(* PLC project Unnamed, Unknown Unnamed 1 *)
(* stored: creationDateTime 2023-04-09T20:23:42, modificationDateTime 2023-05-16T14:21:49 *)

PROGRAM Part1
  VAR_EXTERNAL
    START : BOOL;
    STOP : BOOL;
    CONR4_1 : BOOL;
    CONR4_2 : BOOL;
    SENDIF13 : BOOL;
  END_VAR
  VAR
    SENVIS1 AT %IX100.2 : BOOL;
    SENVIS2 AT %IX100.3 : BOOL;
    SENVIS3 AT %IX100.4 : BOOL;
    SENCAP2 AT %IX102.2 : BOOL;
    SENCAP3 AT %IX102.3 : BOOL;
    SENCAP5 AT %IX102.5 : BOOL;
    SENCAP6 AT %IX102.6 : BOOL;
    TTFrontLimit1 AT %IX103.0 : BOOL;
    TTFrontLimit2 AT %IX103.1 : BOOL;
    TTLimit90_1 AT %IX103.2 : BOOL;
    TTLimit90_2 AT %IX103.3 : BOOL;
    SENCAP8 AT %IX103.4 : BOOL;
    SENCAP9 AT %IX103.5 : BOOL;
    SENCAP10 AT %IX105.1 : BOOL;
    SENCAP11 AT %IX105.2 : BOOL;
    SENCAP12 AT %IX105.3 : BOOL;
    SENCAP13 AT %IX105.4 : BOOL;
    CON2_1 AT %QX100.0 : BOOL;
    CON2_2 AT %QX100.1 : BOOL;
    CON4_1 AT %QX100.2 : BOOL;
    CON4_2 AT %QX100.3 : BOOL;
    CON4_3 AT %QX100.4 : BOOL;
    CON6_1 AT %QX101.0 : BOOL;
    CON6_2 AT %QX101.1 : BOOL;
  END_VAR
  VAR_OUTPUT
    CON6_3 : BOOL;
    CON6_5 : BOOL;
    CON6_7 : BOOL;
  END_VAR
  VAR
    CONSCALE1 AT %QX102.0 : BOOL;
    CONSCALE2 AT %QX102.1 : BOOL;
    CONCURV1 AT %QX102.2 : BOOL;
    CONCURV2 AT %QX102.3 : BOOL;
    PIVOTARM1 AT %QX102.4 : BOOL;
    PIVOTARM2 AT %QX102.5 : BOOL;
    PIVOTARM3 AT %QX102.6 : BOOL;
    PIVOTURN1 AT %QX102.7 : BOOL;
    PIVOTURN2 AT %QX103.0 : BOOL;
    PIVOTURN3 AT %QX103.1 : BOOL;
    MCStart1 AT %QX103.2 : BOOL;
    MCStart2 AT %QX103.3 : BOOL;
    MCStart3 AT %QX103.4 : BOOL;
    MCStop1 AT %QX103.5 : BOOL;
    MCStop2 AT %QX103.6 : BOOL;
    MCStop3 AT %QX103.7 : BOOL;
    TurnTable1 AT %QX109.1 : BOOL;
    TurnTable2 AT %QX109.2 : BOOL;
    TTPles1 AT %QX109.3 : BOOL;
    TTPles2 AT %QX109.4 : BOOL;
    RollStop1 AT %QX109.5 : BOOL;
    RollStop2 AT %QX109.6 : BOOL;
    RollStop3 AT %QX109.7 : BOOL;
    RollStop4 AT %QX110.0 : BOOL;
    RollStop5 AT %QX110.1 : BOOL;
    RollStop6 AT %QX110.2 : BOOL;
  END_VAR
  VAR_EXTERNAL
    RollStop7 : BOOL;
  END_VAR
  VAR
    VIR1 AT %QX4.1 : BOOL;
    VIR2 AT %QX4.2 : BOOL;
    VIR10 AT %QX8.4 : BOOL;
    VIR11 AT %QX8.5 : BOOL;
  END_VAR
  VAR
    TOF1 : TOF;
    TOF2 : TOF;
    CTU0 : CTU;
  END_VAR
  VAR  (* added by the conversion: wires and edge detectors of the diagram *)
    R_TRIG1 : R_TRIG;
    R_TRIG2 : R_TRIG;
    R_TRIG3 : R_TRIG;
    R_TRIG4 : R_TRIG;
  END_VAR

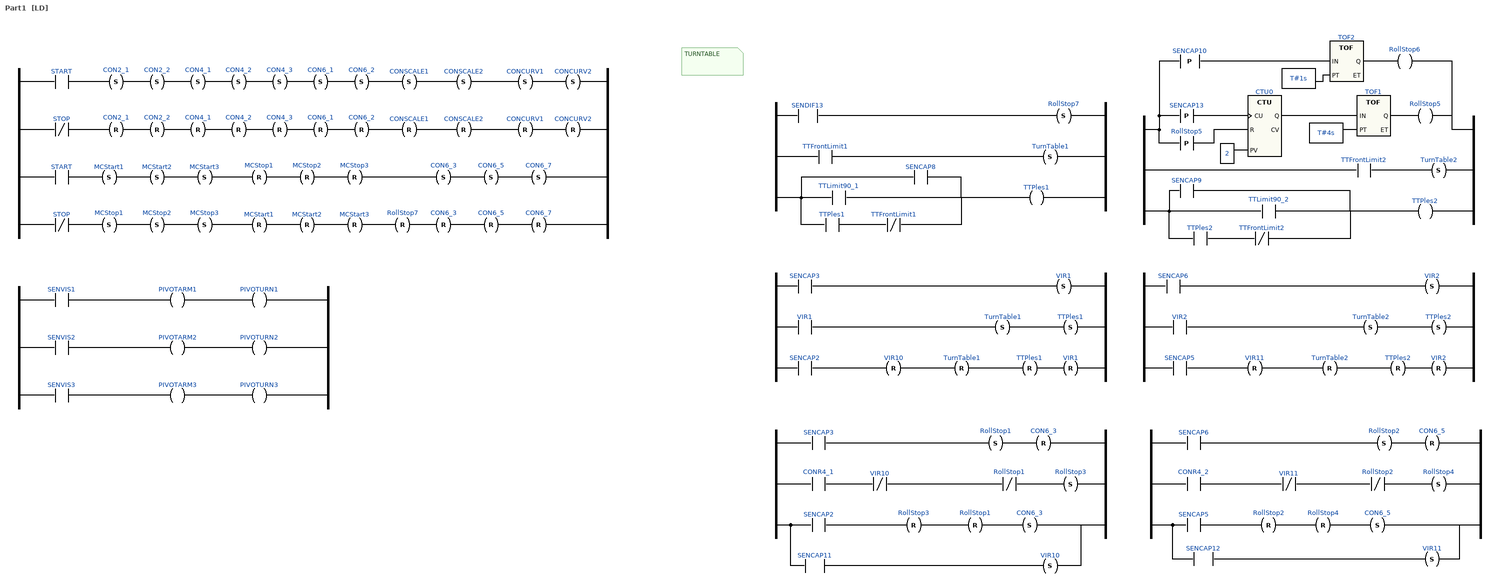
(* LD diagram, written out as Structured Text *)
(* TURNTABLE *)
R_TRIG1(CLK := SENCAP10);
TOF2(IN := R_TRIG1.Q, PT := T#1s);
RollStop6 := TOF2.Q;
IF START THEN CON2_1 := TRUE; END_IF;
IF START THEN CON2_2 := TRUE; END_IF;
IF START THEN CON4_1 := TRUE; END_IF;
IF START THEN CON4_2 := TRUE; END_IF;
IF START THEN CON4_3 := TRUE; END_IF;
IF START THEN CON6_1 := TRUE; END_IF;
IF START THEN CON6_2 := TRUE; END_IF;
IF START THEN CONSCALE1 := TRUE; END_IF;
IF START THEN CONSCALE2 := TRUE; END_IF;
IF START THEN CONCURV1 := TRUE; END_IF;
IF START THEN CONCURV2 := TRUE; END_IF;
IF SENDIF13 THEN RollStop7 := TRUE; END_IF;
R_TRIG2(CLK := SENCAP13);
R_TRIG3(CLK := R_TRIG2.Q);
R_TRIG4(CLK := RollStop5);
CTU0(CU := R_TRIG3.Q, R := R_TRIG4.Q, PV := 2);
TOF1(IN := CTU0.Q, PT := T#4s);
RollStop5 := TOF1.Q;
IF NOT STOP THEN CON2_1 := FALSE; END_IF;
IF NOT STOP THEN CON2_2 := FALSE; END_IF;
IF NOT STOP THEN CON4_1 := FALSE; END_IF;
IF NOT STOP THEN CON4_2 := FALSE; END_IF;
IF NOT STOP THEN CON4_3 := FALSE; END_IF;
IF NOT STOP THEN CON6_1 := FALSE; END_IF;
IF NOT STOP THEN CON6_2 := FALSE; END_IF;
IF NOT STOP THEN CONSCALE1 := FALSE; END_IF;
IF NOT STOP THEN CONSCALE2 := FALSE; END_IF;
IF NOT STOP THEN CONCURV1 := FALSE; END_IF;
IF NOT STOP THEN CONCURV2 := FALSE; END_IF;
IF TTFrontLimit1 THEN TurnTable1 := TRUE; END_IF;
IF TTFrontLimit2 THEN TurnTable2 := TRUE; END_IF;
IF START THEN MCStart1 := TRUE; END_IF;
IF START THEN MCStart2 := TRUE; END_IF;
IF START THEN MCStart3 := TRUE; END_IF;
IF START THEN MCStop1 := FALSE; END_IF;
IF START THEN MCStop2 := FALSE; END_IF;
IF START THEN MCStop3 := FALSE; END_IF;
IF START THEN CON6_3 := TRUE; END_IF;
IF START THEN CON6_5 := TRUE; END_IF;
IF START THEN CON6_7 := TRUE; END_IF;
TTPles1 := TTLimit90_1 OR SENCAP8 OR TTPles1 AND NOT TTFrontLimit1;
TTPles2 := TTLimit90_2 OR SENCAP9 OR TTPles2 AND NOT TTFrontLimit2;
IF NOT STOP THEN MCStop1 := TRUE; END_IF;
IF NOT STOP THEN MCStop2 := TRUE; END_IF;
IF NOT STOP THEN MCStop3 := TRUE; END_IF;
IF NOT STOP THEN MCStart1 := FALSE; END_IF;
IF NOT STOP THEN MCStart2 := FALSE; END_IF;
IF NOT STOP THEN MCStart3 := FALSE; END_IF;
IF NOT STOP THEN RollStop7 := FALSE; END_IF;
IF NOT STOP THEN CON6_3 := FALSE; END_IF;
IF NOT STOP THEN CON6_5 := FALSE; END_IF;
IF NOT STOP THEN CON6_7 := FALSE; END_IF;
IF SENCAP3 THEN VIR1 := TRUE; END_IF;
IF SENCAP6 THEN VIR2 := TRUE; END_IF;
PIVOTARM1 := SENVIS1;
PIVOTURN1 := SENVIS1;
IF VIR1 THEN TurnTable1 := TRUE; END_IF;
IF VIR1 THEN TTPles1 := TRUE; END_IF;
IF VIR2 THEN TurnTable2 := TRUE; END_IF;
IF VIR2 THEN TTPles2 := TRUE; END_IF;
PIVOTARM2 := SENVIS2;
PIVOTURN2 := SENVIS2;
IF SENCAP2 THEN VIR10 := FALSE; END_IF;
IF SENCAP2 THEN TurnTable1 := FALSE; END_IF;
IF SENCAP2 THEN TTPles1 := FALSE; END_IF;
IF SENCAP2 THEN VIR1 := FALSE; END_IF;
IF SENCAP5 THEN VIR11 := FALSE; END_IF;
IF SENCAP5 THEN TurnTable2 := FALSE; END_IF;
IF SENCAP5 THEN TTPles2 := FALSE; END_IF;
IF SENCAP5 THEN VIR2 := FALSE; END_IF;
PIVOTARM3 := SENVIS3;
PIVOTURN3 := SENVIS3;
IF SENCAP3 THEN RollStop1 := TRUE; END_IF;
IF SENCAP3 THEN CON6_3 := FALSE; END_IF;
IF SENCAP6 THEN RollStop2 := TRUE; END_IF;
IF SENCAP6 THEN CON6_5 := FALSE; END_IF;
IF CONR4_1 AND NOT VIR10 AND NOT RollStop1 THEN RollStop3 := TRUE; END_IF;
IF CONR4_2 AND NOT VIR11 AND NOT RollStop2 THEN RollStop4 := TRUE; END_IF;
IF SENCAP2 THEN RollStop3 := FALSE; END_IF;
IF SENCAP2 THEN RollStop1 := FALSE; END_IF;
IF SENCAP2 THEN CON6_3 := TRUE; END_IF;
IF SENCAP5 THEN RollStop2 := FALSE; END_IF;
IF SENCAP5 THEN RollStop4 := FALSE; END_IF;
IF SENCAP5 THEN CON6_5 := TRUE; END_IF;
IF SENCAP12 THEN VIR11 := TRUE; END_IF;
IF SENCAP11 THEN VIR10 := TRUE; END_IF;
END_PROGRAM

PROGRAM Part2
  VAR_EXTERNAL
    START : BOOL;
    STOP : BOOL;
  END_VAR
  VAR
    SENDIF1 AT %IX100.5 : BOOL;
    SENDIF2 AT %IX100.6 : BOOL;
    SENDIF5 AT %IX101.1 : BOOL;
    SENDIF6 AT %IX101.2 : BOOL;
    SENDIF9 AT %IX101.5 : BOOL;
    SENDIF10 AT %IX101.6 : BOOL;
    CON4_4 AT %QX100.5 : BOOL;
    CON4_5 AT %QX100.6 : BOOL;
    CON4_6 AT %QX100.7 : BOOL;
    CLAMP1 AT %QX104.0 : BOOL;
    CLAMP2 AT %QX104.1 : BOOL;
    CLAMP4 AT %QX104.3 : BOOL;
    CLAMP5 AT %QX104.4 : BOOL;
    CLAMP7 AT %QX104.6 : BOOL;
    CLAMP8 AT %QX104.7 : BOOL;
    RiseCLP1 AT %QX105.1 : BOOL;
    RiseCLP4 AT %QX105.2 : BOOL;
    RiseCLP7 AT %QX105.3 : BOOL;
    X1 AT %QX105.4 : BOOL;
    Z1 AT %QX105.5 : BOOL;
    GRAB1 AT %QX105.6 : BOOL;
    X2 AT %QX105.7 : BOOL;
    Z2 AT %QX106.0 : BOOL;
    GRAB2 AT %QX106.1 : BOOL;
    X3 AT %QX106.2 : BOOL;
    Z3 AT %QX106.3 : BOOL;
    GRAB3 AT %QX106.4 : BOOL;
    VIR1 AT %QX0.0 : BOOL;
    VIR2 AT %QX0.1 : BOOL;
    VIR3 AT %QX0.2 : BOOL;
    VIR4 AT %QX0.3 : BOOL;
    VIR5 AT %QX0.4 : BOOL;
    VIR6 AT %QX0.5 : BOOL;
    VIR7 AT %QX0.6 : BOOL;
    VIR8 AT %QX0.7 : BOOL;
    VIR9 AT %QX1.0 : BOOL;
    VIR10 AT %QX1.1 : BOOL;
    VIR11 AT %QX1.2 : BOOL;
    VIR12 AT %QX1.3 : BOOL;
  END_VAR
  VAR
    TON1 : TON;
    TON2 : TON;
    TON3 : TON;
    TON4 : TON;
    TON5 : TON;
    TON0 : TON;
    TON6 : TON;
    TON7 : TON;
    TON8 : TON;
    TON9 : TON;
    TON10 : TON;
    TON11 : TON;
    TON12 : TON;
    TON13 : TON;
    TON14 : TON;
    TON15 : TON;
    TON16 : TON;
    TON17 : TON;
    TON18 : TON;
    TON19 : TON;
    TON20 : TON;
  END_VAR

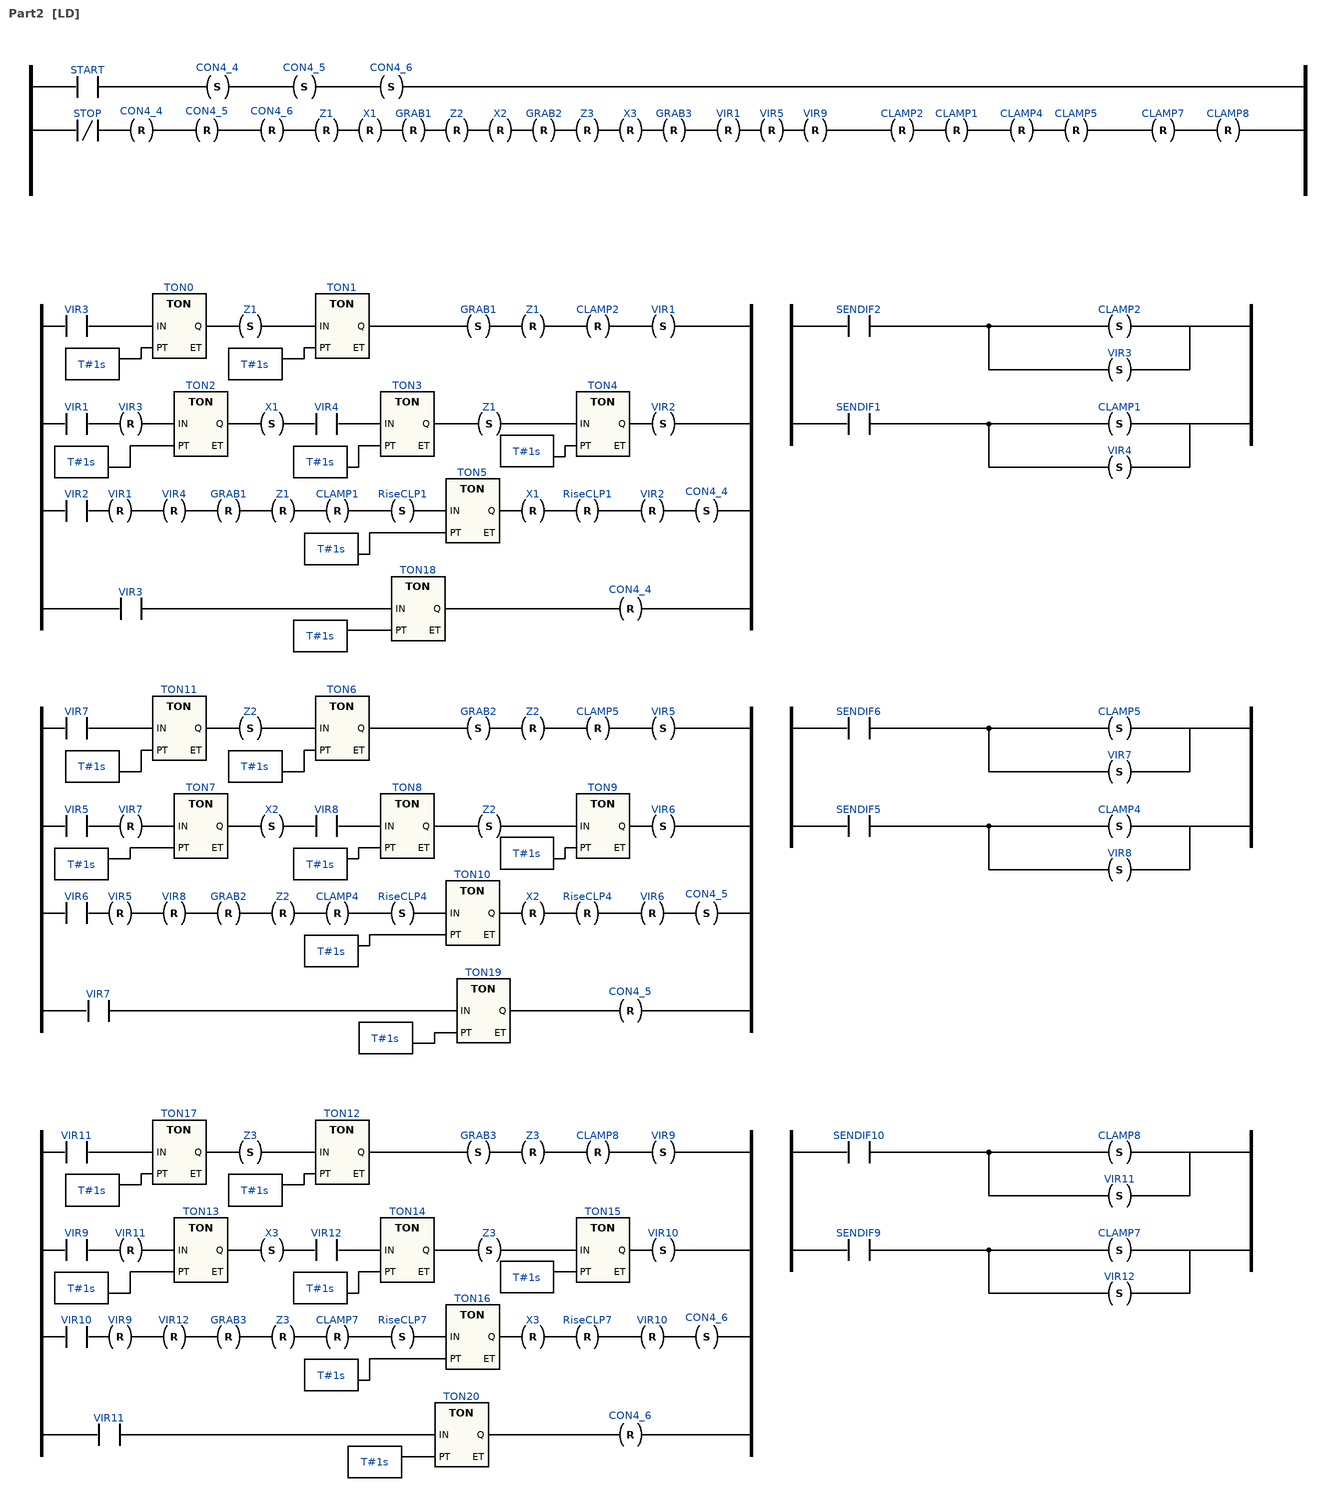
(* LD diagram, written out as Structured Text *)
IF START THEN CON4_4 := TRUE; END_IF;
IF START THEN CON4_5 := TRUE; END_IF;
IF START THEN CON4_6 := TRUE; END_IF;
IF NOT STOP THEN CON4_4 := FALSE; END_IF;
IF NOT STOP THEN CON4_5 := FALSE; END_IF;
IF NOT STOP THEN CON4_6 := FALSE; END_IF;
IF NOT STOP THEN Z1 := FALSE; END_IF;
IF NOT STOP THEN X1 := FALSE; END_IF;
IF NOT STOP THEN GRAB1 := FALSE; END_IF;
IF NOT STOP THEN Z2 := FALSE; END_IF;
IF NOT STOP THEN X2 := FALSE; END_IF;
IF NOT STOP THEN GRAB2 := FALSE; END_IF;
IF NOT STOP THEN Z3 := FALSE; END_IF;
IF NOT STOP THEN X3 := FALSE; END_IF;
IF NOT STOP THEN GRAB3 := FALSE; END_IF;
IF NOT STOP THEN VIR1 := FALSE; END_IF;
IF NOT STOP THEN VIR5 := FALSE; END_IF;
IF NOT STOP THEN VIR9 := FALSE; END_IF;
IF NOT STOP THEN CLAMP2 := FALSE; END_IF;
IF NOT STOP THEN CLAMP1 := FALSE; END_IF;
IF NOT STOP THEN CLAMP4 := FALSE; END_IF;
IF NOT STOP THEN CLAMP5 := FALSE; END_IF;
IF NOT STOP THEN CLAMP7 := FALSE; END_IF;
IF NOT STOP THEN CLAMP8 := FALSE; END_IF;
TON0(IN := VIR3, PT := T#1s);
IF TON0.Q THEN Z1 := TRUE; END_IF;
TON1(IN := TON0.Q, PT := T#1s);
IF TON1.Q THEN GRAB1 := TRUE; END_IF;
IF TON1.Q THEN Z1 := FALSE; END_IF;
IF TON1.Q THEN CLAMP2 := FALSE; END_IF;
IF TON1.Q THEN VIR1 := TRUE; END_IF;
IF SENDIF2 THEN CLAMP2 := TRUE; END_IF;
IF SENDIF2 THEN VIR3 := TRUE; END_IF;
IF VIR1 THEN VIR3 := FALSE; END_IF;
TON2(IN := VIR1, PT := T#1s);
IF TON2.Q THEN X1 := TRUE; END_IF;
TON3(IN := TON2.Q AND VIR4, PT := T#1s);
IF TON3.Q THEN Z1 := TRUE; END_IF;
TON4(IN := TON3.Q, PT := T#1s);
IF TON4.Q THEN VIR2 := TRUE; END_IF;
IF SENDIF1 THEN CLAMP1 := TRUE; END_IF;
IF SENDIF1 THEN VIR4 := TRUE; END_IF;
IF VIR2 THEN VIR1 := FALSE; END_IF;
IF VIR2 THEN VIR4 := FALSE; END_IF;
IF VIR2 THEN GRAB1 := FALSE; END_IF;
IF VIR2 THEN Z1 := FALSE; END_IF;
IF VIR2 THEN CLAMP1 := FALSE; END_IF;
IF VIR2 THEN RiseCLP1 := TRUE; END_IF;
TON5(IN := VIR2, PT := T#1s);
IF TON5.Q THEN X1 := FALSE; END_IF;
IF TON5.Q THEN RiseCLP1 := FALSE; END_IF;
IF TON5.Q THEN VIR2 := FALSE; END_IF;
IF TON5.Q THEN CON4_4 := TRUE; END_IF;
TON18(IN := VIR3, PT := T#1s);
IF TON18.Q THEN CON4_4 := FALSE; END_IF;
TON11(IN := VIR7, PT := T#1s);
IF TON11.Q THEN Z2 := TRUE; END_IF;
TON6(IN := TON11.Q, PT := T#1s);
IF TON6.Q THEN GRAB2 := TRUE; END_IF;
IF TON6.Q THEN Z2 := FALSE; END_IF;
IF TON6.Q THEN CLAMP5 := FALSE; END_IF;
IF TON6.Q THEN VIR5 := TRUE; END_IF;
IF SENDIF6 THEN CLAMP5 := TRUE; END_IF;
IF SENDIF6 THEN VIR7 := TRUE; END_IF;
IF VIR5 THEN VIR7 := FALSE; END_IF;
TON7(IN := VIR5, PT := T#1s);
IF TON7.Q THEN X2 := TRUE; END_IF;
TON8(IN := TON7.Q AND VIR8, PT := T#1s);
IF TON8.Q THEN Z2 := TRUE; END_IF;
TON9(IN := TON8.Q, PT := T#1s);
IF TON9.Q THEN VIR6 := TRUE; END_IF;
IF SENDIF5 THEN CLAMP4 := TRUE; END_IF;
IF SENDIF5 THEN VIR8 := TRUE; END_IF;
IF VIR6 THEN VIR5 := FALSE; END_IF;
IF VIR6 THEN VIR8 := FALSE; END_IF;
IF VIR6 THEN GRAB2 := FALSE; END_IF;
IF VIR6 THEN Z2 := FALSE; END_IF;
IF VIR6 THEN CLAMP4 := FALSE; END_IF;
IF VIR6 THEN RiseCLP4 := TRUE; END_IF;
TON10(IN := VIR6, PT := T#1s);
IF TON10.Q THEN X2 := FALSE; END_IF;
IF TON10.Q THEN RiseCLP4 := FALSE; END_IF;
IF TON10.Q THEN VIR6 := FALSE; END_IF;
IF TON10.Q THEN CON4_5 := TRUE; END_IF;
TON19(IN := VIR7, PT := T#1s);
IF TON19.Q THEN CON4_5 := FALSE; END_IF;
TON17(IN := VIR11, PT := T#1s);
IF TON17.Q THEN Z3 := TRUE; END_IF;
TON12(IN := TON17.Q, PT := T#1s);
IF TON12.Q THEN GRAB3 := TRUE; END_IF;
IF TON12.Q THEN Z3 := FALSE; END_IF;
IF TON12.Q THEN CLAMP8 := FALSE; END_IF;
IF TON12.Q THEN VIR9 := TRUE; END_IF;
IF SENDIF10 THEN CLAMP8 := TRUE; END_IF;
IF SENDIF10 THEN VIR11 := TRUE; END_IF;
IF VIR9 THEN VIR11 := FALSE; END_IF;
TON13(IN := VIR9, PT := T#1s);
IF TON13.Q THEN X3 := TRUE; END_IF;
TON14(IN := TON13.Q AND VIR12, PT := T#1s);
IF TON14.Q THEN Z3 := TRUE; END_IF;
TON15(IN := TON14.Q, PT := T#1s);
IF TON15.Q THEN VIR10 := TRUE; END_IF;
IF SENDIF9 THEN CLAMP7 := TRUE; END_IF;
IF SENDIF9 THEN VIR12 := TRUE; END_IF;
IF VIR10 THEN VIR9 := FALSE; END_IF;
IF VIR10 THEN VIR12 := FALSE; END_IF;
IF VIR10 THEN GRAB3 := FALSE; END_IF;
IF VIR10 THEN Z3 := FALSE; END_IF;
IF VIR10 THEN CLAMP7 := FALSE; END_IF;
IF VIR10 THEN RiseCLP7 := TRUE; END_IF;
TON16(IN := VIR10, PT := T#1s);
IF TON16.Q THEN X3 := FALSE; END_IF;
IF TON16.Q THEN RiseCLP7 := FALSE; END_IF;
IF TON16.Q THEN VIR10 := FALSE; END_IF;
IF TON16.Q THEN CON4_6 := TRUE; END_IF;
TON20(IN := VIR11, PT := T#1s);
IF TON20.Q THEN CON4_6 := FALSE; END_IF;
END_PROGRAM

PROGRAM Part3
  VAR_EXTERNAL
    START : BOOL;
    STOP : BOOL;
  END_VAR
  VAR
    SENDIF3 AT %IX100.7 : BOOL;
    SENDIF4 AT %IX101.0 : BOOL;
    SENDIF7 AT %IX101.3 : BOOL;
    SENDIF8 AT %IX101.4 : BOOL;
    SENDIF11 AT %IX101.7 : BOOL;
    SENDIF12 AT %IX102.0 : BOOL;
    SENCAP1 AT %IX102.1 : BOOL;
    SENCAP4 AT %IX102.4 : BOOL;
    SENCAP7 AT %IX102.7 : BOOL;
    CON6_4 AT %QX101.3 : BOOL;
    CON6_6 AT %QX101.5 : BOOL;
    CON6_8 AT %QX101.7 : BOOL;
    CLAMP3 AT %QX104.2 : BOOL;
    CLAMP6 AT %QX104.5 : BOOL;
    CLAMP9 AT %QX105.0 : BOOL;
    CW4 AT %QX106.5 : BOOL;
    CCW4 AT %QX106.6 : BOOL;
    CW5 AT %QX106.7 : BOOL;
    CCW5 AT %QX107.0 : BOOL;
    CW6 AT %QX107.1 : BOOL;
    CCW6 AT %QX107.2 : BOOL;
    GRAB4 AT %QX107.3 : BOOL;
    GRAB5 AT %QX107.4 : BOOL;
    GRAB6 AT %QX107.5 : BOOL;
    CONR2_1 AT %QX107.6 : BOOL;
    CONR2_2 AT %QX107.7 : BOOL;
    CONR2_3 AT %QX108.0 : BOOL;
  END_VAR
  VAR_EXTERNAL
    CONR4_1 : BOOL;
    CONR4_2 : BOOL;
  END_VAR
  VAR
    CONR4_3 AT %QX108.3 : BOOL;
    CONR4_4 AT %QX108.4 : BOOL;
    CONR6_1 AT %QX108.5 : BOOL;
    CONR6_2 AT %QX108.6 : BOOL;
    CONRLCCW1 AT %QX108.7 : BOOL;
    CONRLCCW2 AT %QX109.0 : BOOL;
    CLPRise3 AT %QX112.2 : BOOL;
    CLPRise6 AT %QX112.3 : BOOL;
    CLPRise9 AT %QX112.4 : BOOL;
    X4 AT %QW100 : INT;
    Z4 AT %QW101 : INT;
    X5 AT %QW102 : INT;
    Z5 AT %QW103 : INT;
    X6 AT %QW104 : INT;
    Z6 AT %QW105 : INT;
    VIR1 AT %QX1.4 : BOOL;
    VIR2 AT %QX1.5 : BOOL;
    VIR3 AT %QX1.6 : BOOL;
    VIR4 AT %QX1.7 : BOOL;
    VIR5 AT %QX2.0 : BOOL;
    VIR6 AT %QX2.1 : BOOL;
    VIR7 AT %QX2.2 : BOOL;
    VIR8 AT %QX2.3 : BOOL;
    VIR9 AT %QX2.4 : BOOL;
    VIR10 AT %QX2.5 : BOOL;
    VIR11 AT %QX2.6 : BOOL;
    VIR12 AT %QX2.7 : BOOL;
    VIR13 AT %QX3.0 : BOOL;
    VIR14 AT %QX3.1 : BOOL;
    VIR15 AT %QX3.2 : BOOL;
    VIR16 AT %QX3.3 : BOOL;
    VIR17 AT %QX3.4 : BOOL;
    VIR18 AT %QX3.5 : BOOL;
    VIR19 AT %QX3.6 : BOOL;
    VIR20 AT %QX3.7 : BOOL;
    VIR21 AT %QX4.0 : BOOL;
    VIR22 AT %QX5.6 : BOOL;
    VIR23 AT %QX5.7 : BOOL;
  END_VAR
  VAR_EXTERNAL
    CON6_3 : BOOL;
    CON6_5 : BOOL;
    CON6_7 : BOOL;
  END_VAR
  VAR
    TON0 : TON;
    TON1 : TON;
    TON2 : TON;
    TON3 : TON;
    TON4 : TON;
    TON5 : TON;
    TON6 : TON;
    TON7 : TON;
    TON8 : TON;
    TON9 : TON;
    TON10 : TON;
    TON11 : TON;
    TON12 : TON;
    TON13 : TON;
    TON14 : TON;
    TON15 : TON;
    TON16 : TON;
    CTU0 : CTU;
    TON17 : TON;
    TON18 : TON;
    TON19 : TON;
    TON20 : TON;
    TON21 : TON;
    TON22 : TON;
    TON23 : TON;
    TON24 : TON;
    TON25 : TON;
    TON26 : TON;
    TON27 : TON;
    TON28 : TON;
    TON29 : TON;
    TON30 : TON;
    TON31 : TON;
    TON32 : TON;
    TON33 : TON;
    CTU1 : CTU;
    TON34 : TON;
    TON35 : TON;
    TON36 : TON;
    TON37 : TON;
    TON38 : TON;
    TON39 : TON;
    TON40 : TON;
    TON41 : TON;
    TON42 : TON;
    TON43 : TON;
    TON44 : TON;
    TON45 : TON;
    TON46 : TON;
    TON47 : TON;
    TON48 : TON;
    TON49 : TON;
    TON50 : TON;
    CTU2 : CTU;
    TON51 : TON;
    TON52 : TON;
    TON53 : TON;
  END_VAR
  VAR  (* added by the conversion: wires and edge detectors of the diagram *)
    _MOVE66_ENO : BOOL;
    _MOVE66_OUT : INT;
    _MOVE25_ENO : BOOL;
    _MOVE25_OUT : INT;
    _MOVE288_ENO : BOOL;
    _MOVE288_OUT : INT;
    _MOVE249_ENO : BOOL;
    _MOVE249_OUT : INT;
    _MOVE44_ENO : BOOL;
    _MOVE44_OUT : INT;
    _MOVE51_ENO : BOOL;
    _MOVE51_OUT : INT;
    _MOVE268_ENO : BOOL;
    _MOVE268_OUT : INT;
    _MOVE275_ENO : BOOL;
    _MOVE275_OUT : INT;
    _MOVE73_ENO : BOOL;
    _MOVE73_OUT : INT;
    _MOVE76_ENO : BOOL;
    _MOVE76_OUT : INT;
    _MOVE83_ENO : BOOL;
    _MOVE83_OUT : INT;
    _MOVE295_ENO : BOOL;
    _MOVE295_OUT : INT;
    _MOVE298_ENO : BOOL;
    _MOVE298_OUT : INT;
    _MOVE305_ENO : BOOL;
    _MOVE305_OUT : INT;
    _MOVE89_ENO : BOOL;
    _MOVE89_OUT : INT;
    _MOVE94_ENO : BOOL;
    _MOVE94_OUT : INT;
    _MOVE311_ENO : BOOL;
    _MOVE311_OUT : INT;
    _MOVE316_ENO : BOOL;
    _MOVE316_OUT : INT;
    _MOVE100_ENO : BOOL;
    _MOVE100_OUT : INT;
    _MOVE322_ENO : BOOL;
    _MOVE322_OUT : INT;
    R_TRIG1 : R_TRIG;
    R_TRIG2 : R_TRIG;
    _MOVE177_ENO : BOOL;
    _MOVE177_OUT : INT;
    _MOVE138_ENO : BOOL;
    _MOVE138_OUT : INT;
    _MOVE157_ENO : BOOL;
    _MOVE157_OUT : INT;
    _MOVE164_ENO : BOOL;
    _MOVE164_OUT : INT;
    _MOVE184_ENO : BOOL;
    _MOVE184_OUT : INT;
    _MOVE187_ENO : BOOL;
    _MOVE187_OUT : INT;
    _MOVE194_ENO : BOOL;
    _MOVE194_OUT : INT;
    _MOVE200_ENO : BOOL;
    _MOVE200_OUT : INT;
    _MOVE205_ENO : BOOL;
    _MOVE205_OUT : INT;
    _MOVE211_ENO : BOOL;
    _MOVE211_OUT : INT;
    R_TRIG3 : R_TRIG;
  END_VAR

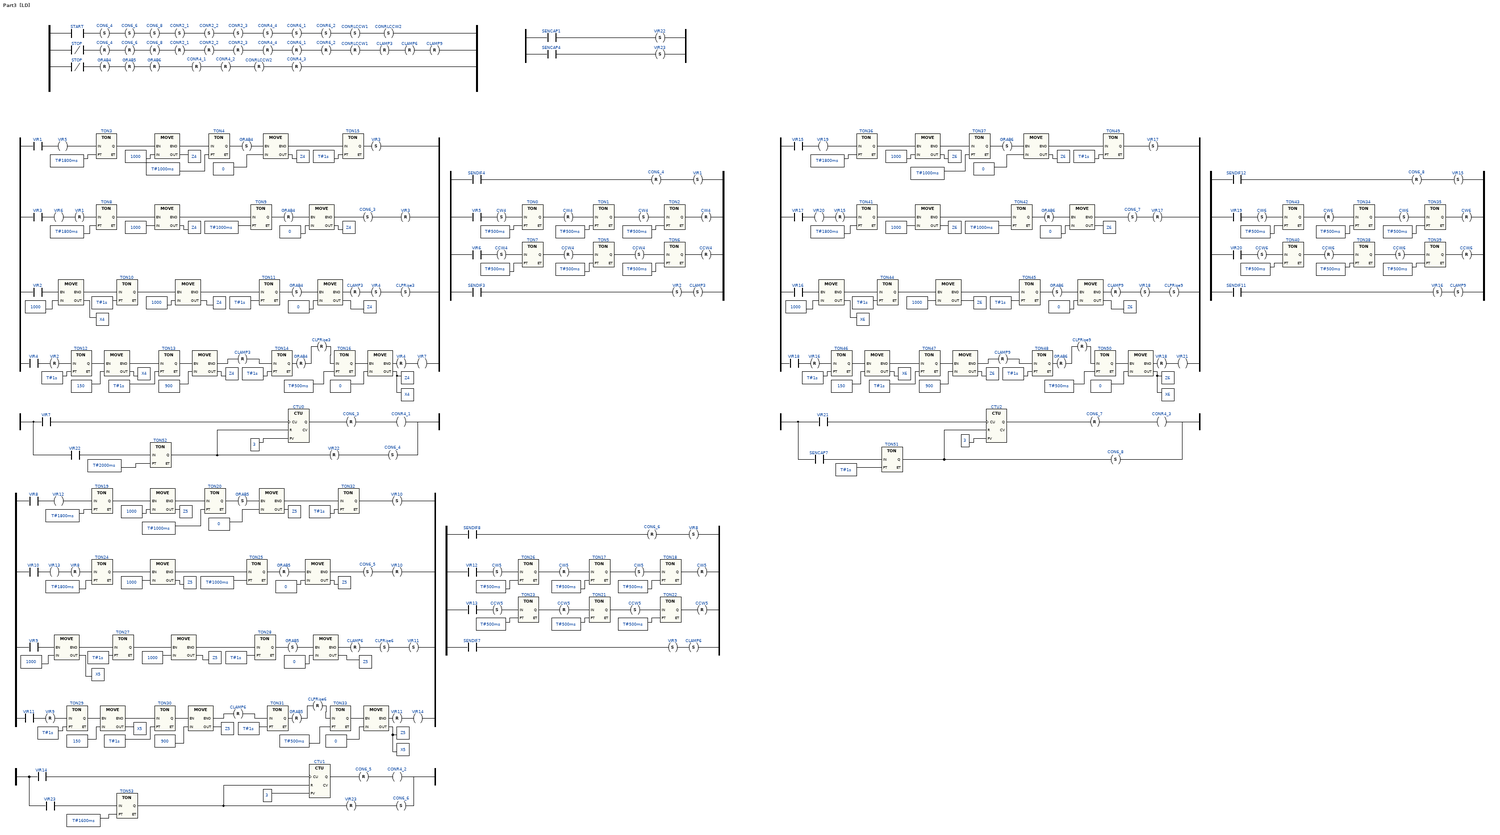
(* LD diagram, written out as Structured Text *)
IF START THEN CON6_4 := TRUE; END_IF;
IF START THEN CON6_6 := TRUE; END_IF;
IF START THEN CON6_8 := TRUE; END_IF;
IF START THEN CONR2_1 := TRUE; END_IF;
IF START THEN CONR2_2 := TRUE; END_IF;
IF START THEN CONR2_3 := TRUE; END_IF;
IF START THEN CONR4_4 := TRUE; END_IF;
IF START THEN CONR6_1 := TRUE; END_IF;
IF START THEN CONR6_2 := TRUE; END_IF;
IF START THEN CONRLCCW1 := TRUE; END_IF;
IF START THEN CONRLCCW2 := TRUE; END_IF;
IF SENCAP1 THEN VIR22 := TRUE; END_IF;
IF NOT STOP THEN CON6_4 := FALSE; END_IF;
IF NOT STOP THEN CON6_6 := FALSE; END_IF;
IF NOT STOP THEN CON6_8 := FALSE; END_IF;
IF NOT STOP THEN CONR2_1 := FALSE; END_IF;
IF NOT STOP THEN CONR2_2 := FALSE; END_IF;
IF NOT STOP THEN CONR2_3 := FALSE; END_IF;
IF NOT STOP THEN CONR4_4 := FALSE; END_IF;
IF NOT STOP THEN CONR6_1 := FALSE; END_IF;
IF NOT STOP THEN CONR6_2 := FALSE; END_IF;
IF NOT STOP THEN CONRLCCW1 := FALSE; END_IF;
IF NOT STOP THEN CLAMP3 := FALSE; END_IF;
IF NOT STOP THEN CLAMP6 := FALSE; END_IF;
IF NOT STOP THEN CLAMP9 := FALSE; END_IF;
IF SENCAP4 THEN VIR23 := TRUE; END_IF;
IF NOT STOP THEN GRAB4 := FALSE; END_IF;
IF NOT STOP THEN GRAB5 := FALSE; END_IF;
IF NOT STOP THEN GRAB6 := FALSE; END_IF;
IF NOT STOP THEN CONR4_1 := FALSE; END_IF;
IF NOT STOP THEN CONR4_2 := FALSE; END_IF;
IF NOT STOP THEN CONRLCCW2 := FALSE; END_IF;
IF NOT STOP THEN CONR4_3 := FALSE; END_IF;
VIR5 := VIR1;
TON3(IN := VIR1, PT := T#1800ms);
_MOVE66_OUT := MOVE(EN := TON3.Q, IN := 1000, ENO => _MOVE66_ENO);
TON4(IN := _MOVE66_ENO, PT := T#1000ms);
IF TON4.Q THEN GRAB4 := TRUE; END_IF;
_MOVE25_OUT := MOVE(EN := TON4.Q, IN := 0, ENO => _MOVE25_ENO);
TON15(IN := _MOVE25_ENO, PT := T#1s);
IF TON15.Q THEN VIR3 := TRUE; END_IF;
VIR19 := VIR15;
TON36(IN := VIR15, PT := T#1800ms);
_MOVE288_OUT := MOVE(EN := TON36.Q, IN := 1000, ENO => _MOVE288_ENO);
TON37(IN := _MOVE288_ENO, PT := T#1000ms);
IF TON37.Q THEN GRAB6 := TRUE; END_IF;
_MOVE249_OUT := MOVE(EN := TON37.Q, IN := 0, ENO => _MOVE249_ENO);
TON49(IN := _MOVE249_ENO, PT := T#1s);
IF TON49.Q THEN VIR17 := TRUE; END_IF;
IF _MOVE66_ENO THEN Z4 := _MOVE66_OUT; END_IF;
IF _MOVE25_ENO THEN Z4 := _MOVE25_OUT; END_IF;
IF _MOVE288_ENO THEN Z6 := _MOVE288_OUT; END_IF;
IF _MOVE249_ENO THEN Z6 := _MOVE249_OUT; END_IF;
IF SENDIF4 THEN CON6_4 := FALSE; END_IF;
IF SENDIF4 THEN VIR1 := TRUE; END_IF;
IF SENDIF12 THEN CON6_8 := FALSE; END_IF;
IF SENDIF12 THEN VIR15 := TRUE; END_IF;
VIR6 := VIR3;
IF VIR3 THEN VIR1 := FALSE; END_IF;
TON8(IN := VIR3, PT := T#1800ms);
_MOVE44_OUT := MOVE(EN := TON8.Q, IN := 1000, ENO => _MOVE44_ENO);
TON9(IN := _MOVE44_ENO, PT := T#1000ms);
IF TON9.Q THEN GRAB4 := FALSE; END_IF;
_MOVE51_OUT := MOVE(EN := TON9.Q, IN := 0, ENO => _MOVE51_ENO);
IF _MOVE51_ENO THEN CON6_3 := TRUE; END_IF;
IF _MOVE51_ENO THEN VIR3 := FALSE; END_IF;
IF VIR5 THEN CW4 := TRUE; END_IF;
TON0(IN := VIR5, PT := T#500ms);
IF TON0.Q THEN CW4 := FALSE; END_IF;
TON1(IN := TON0.Q, PT := T#500ms);
IF TON1.Q THEN CW4 := TRUE; END_IF;
TON2(IN := TON1.Q, PT := T#500ms);
IF TON2.Q THEN CW4 := FALSE; END_IF;
VIR20 := VIR17;
IF VIR17 THEN VIR15 := FALSE; END_IF;
TON41(IN := VIR17, PT := T#1800ms);
_MOVE268_OUT := MOVE(EN := TON41.Q, IN := 1000, ENO => _MOVE268_ENO);
TON42(IN := _MOVE268_ENO, PT := T#1000ms);
IF TON42.Q THEN GRAB6 := FALSE; END_IF;
_MOVE275_OUT := MOVE(EN := TON42.Q, IN := 0, ENO => _MOVE275_ENO);
IF _MOVE275_ENO THEN CON6_7 := TRUE; END_IF;
IF _MOVE275_ENO THEN VIR17 := FALSE; END_IF;
IF VIR19 THEN CW6 := TRUE; END_IF;
TON43(IN := VIR19, PT := T#500ms);
IF TON43.Q THEN CW6 := FALSE; END_IF;
TON34(IN := TON43.Q, PT := T#500ms);
IF TON34.Q THEN CW6 := TRUE; END_IF;
TON35(IN := TON34.Q, PT := T#500ms);
IF TON35.Q THEN CW6 := FALSE; END_IF;
IF _MOVE44_ENO THEN Z4 := _MOVE44_OUT; END_IF;
IF _MOVE51_ENO THEN Z4 := _MOVE51_OUT; END_IF;
IF _MOVE268_ENO THEN Z6 := _MOVE268_OUT; END_IF;
IF _MOVE275_ENO THEN Z6 := _MOVE275_OUT; END_IF;
IF VIR6 THEN CCW4 := TRUE; END_IF;
TON7(IN := VIR6, PT := T#500ms);
IF TON7.Q THEN CCW4 := FALSE; END_IF;
TON5(IN := TON7.Q, PT := T#500ms);
IF TON5.Q THEN CCW4 := TRUE; END_IF;
TON6(IN := TON5.Q, PT := T#500ms);
IF TON6.Q THEN CCW4 := FALSE; END_IF;
IF VIR20 THEN CCW6 := TRUE; END_IF;
TON40(IN := VIR20, PT := T#500ms);
IF TON40.Q THEN CCW6 := FALSE; END_IF;
TON38(IN := TON40.Q, PT := T#500ms);
IF TON38.Q THEN CCW6 := TRUE; END_IF;
TON39(IN := TON38.Q, PT := T#500ms);
IF TON39.Q THEN CCW6 := FALSE; END_IF;
_MOVE73_OUT := MOVE(EN := VIR2, IN := 1000, ENO => _MOVE73_ENO);
TON10(IN := _MOVE73_ENO, PT := T#1s);
_MOVE76_OUT := MOVE(EN := TON10.Q, IN := 1000, ENO => _MOVE76_ENO);
TON11(IN := _MOVE76_ENO, PT := T#1s);
IF TON11.Q THEN GRAB4 := TRUE; END_IF;
_MOVE83_OUT := MOVE(EN := TON11.Q, IN := 0, ENO => _MOVE83_ENO);
IF _MOVE83_ENO THEN CLAMP3 := FALSE; END_IF;
IF _MOVE83_ENO THEN VIR4 := TRUE; END_IF;
IF _MOVE83_ENO THEN CLPRise3 := TRUE; END_IF;
IF SENDIF3 THEN VIR2 := TRUE; END_IF;
IF SENDIF3 THEN CLAMP3 := TRUE; END_IF;
_MOVE295_OUT := MOVE(EN := VIR16, IN := 1000, ENO => _MOVE295_ENO);
TON44(IN := _MOVE295_ENO, PT := T#1s);
_MOVE298_OUT := MOVE(EN := TON44.Q, IN := 1000, ENO => _MOVE298_ENO);
TON45(IN := _MOVE298_ENO, PT := T#1s);
IF TON45.Q THEN GRAB6 := TRUE; END_IF;
_MOVE305_OUT := MOVE(EN := TON45.Q, IN := 0, ENO => _MOVE305_ENO);
IF _MOVE305_ENO THEN CLAMP9 := FALSE; END_IF;
IF _MOVE305_ENO THEN VIR18 := TRUE; END_IF;
IF _MOVE305_ENO THEN CLPRise9 := TRUE; END_IF;
IF SENDIF11 THEN VIR16 := TRUE; END_IF;
IF SENDIF11 THEN CLAMP9 := TRUE; END_IF;
IF _MOVE76_ENO THEN Z4 := _MOVE76_OUT; END_IF;
IF _MOVE298_ENO THEN Z6 := _MOVE298_OUT; END_IF;
IF _MOVE83_ENO THEN Z4 := _MOVE83_OUT; END_IF;
IF _MOVE305_ENO THEN Z6 := _MOVE305_OUT; END_IF;
IF _MOVE73_ENO THEN X4 := _MOVE73_OUT; END_IF;
IF _MOVE295_ENO THEN X6 := _MOVE295_OUT; END_IF;
TON12(IN := VIR4, PT := T#1s);
_MOVE89_OUT := MOVE(EN := TON12.Q, IN := 150, ENO => _MOVE89_ENO);
TON13(IN := _MOVE89_ENO, PT := T#1s);
_MOVE94_OUT := MOVE(EN := TON13.Q, IN := 900, ENO => _MOVE94_ENO);
TON14(IN := _MOVE94_ENO, PT := T#1s);
IF TON14.Q THEN CLPRise3 := FALSE; END_IF;
TON46(IN := VIR18, PT := T#1s);
_MOVE311_OUT := MOVE(EN := TON46.Q, IN := 150, ENO => _MOVE311_ENO);
TON47(IN := _MOVE311_ENO, PT := T#1s);
_MOVE316_OUT := MOVE(EN := TON47.Q, IN := 900, ENO => _MOVE316_ENO);
TON48(IN := _MOVE316_ENO, PT := T#1s);
IF TON48.Q THEN CLPRise9 := FALSE; END_IF;
IF _MOVE94_ENO THEN CLAMP3 := FALSE; END_IF;
IF _MOVE316_ENO THEN CLAMP9 := FALSE; END_IF;
IF VIR4 THEN VIR2 := FALSE; END_IF;
IF TON14.Q THEN GRAB4 := FALSE; END_IF;
TON16(IN := TON14.Q, PT := T#500ms);
_MOVE100_OUT := MOVE(EN := TON16.Q, IN := 0, ENO => _MOVE100_ENO);
IF _MOVE100_ENO THEN VIR4 := FALSE; END_IF;
VIR7 := _MOVE100_ENO;
IF VIR18 THEN VIR16 := FALSE; END_IF;
IF TON48.Q THEN GRAB6 := FALSE; END_IF;
TON50(IN := TON48.Q, PT := T#500ms);
_MOVE322_OUT := MOVE(EN := TON50.Q, IN := 0, ENO => _MOVE322_ENO);
IF _MOVE322_ENO THEN VIR18 := FALSE; END_IF;
VIR21 := _MOVE322_ENO;
IF _MOVE89_ENO THEN X4 := _MOVE89_OUT; END_IF;
IF _MOVE94_ENO THEN Z4 := _MOVE94_OUT; END_IF;
IF _MOVE311_ENO THEN X6 := _MOVE311_OUT; END_IF;
IF _MOVE316_ENO THEN Z6 := _MOVE316_OUT; END_IF;
IF _MOVE100_ENO THEN Z4 := _MOVE100_OUT; END_IF;
IF _MOVE322_ENO THEN Z6 := _MOVE322_OUT; END_IF;
IF _MOVE100_ENO THEN X4 := _MOVE100_OUT; END_IF;
IF _MOVE322_ENO THEN X6 := _MOVE322_OUT; END_IF;
R_TRIG1(CLK := VIR7);
TON52(IN := VIR22, PT := T#2000ms);
CTU0(CU := R_TRIG1.Q, R := TON52.Q, PV := 3);
IF CTU0.Q THEN CON6_3 := FALSE; END_IF;
CONR4_1 := CTU0.Q;
R_TRIG2(CLK := VIR21);
TON51(IN := SENCAP7, PT := T#1s);
CTU2(CU := R_TRIG2.Q, R := TON51.Q, PV := 3);
IF CTU2.Q THEN CON6_7 := FALSE; END_IF;
CONR4_3 := CTU2.Q;
IF TON52.Q THEN VIR22 := FALSE; END_IF;
IF TON52.Q THEN CON6_4 := TRUE; END_IF;
IF TON51.Q THEN CON6_8 := TRUE; END_IF;
VIR12 := VIR8;
TON19(IN := VIR8, PT := T#1800ms);
_MOVE177_OUT := MOVE(EN := TON19.Q, IN := 1000, ENO => _MOVE177_ENO);
TON20(IN := _MOVE177_ENO, PT := T#1000ms);
IF TON20.Q THEN GRAB5 := TRUE; END_IF;
_MOVE138_OUT := MOVE(EN := TON20.Q, IN := 0, ENO => _MOVE138_ENO);
TON32(IN := _MOVE138_ENO, PT := T#1s);
IF TON32.Q THEN VIR10 := TRUE; END_IF;
IF _MOVE177_ENO THEN Z5 := _MOVE177_OUT; END_IF;
IF _MOVE138_ENO THEN Z5 := _MOVE138_OUT; END_IF;
IF SENDIF8 THEN CON6_6 := FALSE; END_IF;
IF SENDIF8 THEN VIR8 := TRUE; END_IF;
VIR13 := VIR10;
IF VIR10 THEN VIR8 := FALSE; END_IF;
TON24(IN := VIR10, PT := T#1800ms);
_MOVE157_OUT := MOVE(EN := TON24.Q, IN := 1000, ENO => _MOVE157_ENO);
TON25(IN := _MOVE157_ENO, PT := T#1000ms);
IF TON25.Q THEN GRAB5 := FALSE; END_IF;
_MOVE164_OUT := MOVE(EN := TON25.Q, IN := 0, ENO => _MOVE164_ENO);
IF _MOVE164_ENO THEN CON6_5 := TRUE; END_IF;
IF _MOVE164_ENO THEN VIR10 := FALSE; END_IF;
IF VIR12 THEN CW5 := TRUE; END_IF;
TON26(IN := VIR12, PT := T#500ms);
IF TON26.Q THEN CW5 := FALSE; END_IF;
TON17(IN := TON26.Q, PT := T#500ms);
IF TON17.Q THEN CW5 := TRUE; END_IF;
TON18(IN := TON17.Q, PT := T#500ms);
IF TON18.Q THEN CW5 := FALSE; END_IF;
IF _MOVE157_ENO THEN Z5 := _MOVE157_OUT; END_IF;
IF _MOVE164_ENO THEN Z5 := _MOVE164_OUT; END_IF;
IF VIR13 THEN CCW5 := TRUE; END_IF;
TON23(IN := VIR13, PT := T#500ms);
IF TON23.Q THEN CCW5 := FALSE; END_IF;
TON21(IN := TON23.Q, PT := T#500ms);
IF TON21.Q THEN CCW5 := TRUE; END_IF;
TON22(IN := TON21.Q, PT := T#500ms);
IF TON22.Q THEN CCW5 := FALSE; END_IF;
_MOVE184_OUT := MOVE(EN := VIR9, IN := 1000, ENO => _MOVE184_ENO);
TON27(IN := _MOVE184_ENO, PT := T#1s);
_MOVE187_OUT := MOVE(EN := TON27.Q, IN := 1000, ENO => _MOVE187_ENO);
TON28(IN := _MOVE187_ENO, PT := T#1s);
IF TON28.Q THEN GRAB5 := TRUE; END_IF;
_MOVE194_OUT := MOVE(EN := TON28.Q, IN := 0, ENO => _MOVE194_ENO);
IF _MOVE194_ENO THEN CLAMP6 := FALSE; END_IF;
IF _MOVE194_ENO THEN CLPRise6 := TRUE; END_IF;
IF _MOVE194_ENO THEN VIR11 := TRUE; END_IF;
IF SENDIF7 THEN VIR9 := TRUE; END_IF;
IF SENDIF7 THEN CLAMP6 := TRUE; END_IF;
IF _MOVE187_ENO THEN Z5 := _MOVE187_OUT; END_IF;
IF _MOVE194_ENO THEN Z5 := _MOVE194_OUT; END_IF;
IF _MOVE184_ENO THEN X5 := _MOVE184_OUT; END_IF;
TON29(IN := VIR11, PT := T#1s);
_MOVE200_OUT := MOVE(EN := TON29.Q, IN := 150, ENO => _MOVE200_ENO);
TON30(IN := _MOVE200_ENO, PT := T#1s);
_MOVE205_OUT := MOVE(EN := TON30.Q, IN := 900, ENO => _MOVE205_ENO);
TON31(IN := _MOVE205_ENO, PT := T#1s);
IF TON31.Q THEN CLPRise6 := FALSE; END_IF;
IF _MOVE205_ENO THEN CLAMP6 := FALSE; END_IF;
IF VIR11 THEN VIR9 := FALSE; END_IF;
IF TON31.Q THEN GRAB5 := FALSE; END_IF;
TON33(IN := TON31.Q, PT := T#500ms);
_MOVE211_OUT := MOVE(EN := TON33.Q, IN := 0, ENO => _MOVE211_ENO);
IF _MOVE211_ENO THEN VIR11 := FALSE; END_IF;
VIR14 := _MOVE211_ENO;
IF _MOVE200_ENO THEN X5 := _MOVE200_OUT; END_IF;
IF _MOVE205_ENO THEN Z5 := _MOVE205_OUT; END_IF;
IF _MOVE211_ENO THEN Z5 := _MOVE211_OUT; END_IF;
IF _MOVE211_ENO THEN X5 := _MOVE211_OUT; END_IF;
R_TRIG3(CLK := VIR14);
TON53(IN := VIR23, PT := T#1600ms);
CTU1(CU := R_TRIG3.Q, R := TON53.Q, PV := 3);
IF CTU1.Q THEN CON6_5 := FALSE; END_IF;
CONR4_2 := CTU1.Q;
IF TON53.Q THEN VIR23 := FALSE; END_IF;
IF TON53.Q THEN CON6_6 := TRUE; END_IF;
END_PROGRAM

PROGRAM Part4
  VAR_EXTERNAL
    START : BOOL;
    STOP : BOOL;
    SENDIF13 : BOOL;
    RollStop7 : BOOL;
  END_VAR
  VAR
    SENDIF14 AT %IX103.7 : BOOL;
    SENDIF15 AT %IX104.0 : BOOL;
    SENVIS4 AT %IX104.1 : BOOL;
    SENVIS5 AT %IX104.2 : BOOL;
    X1 AT %IX104.3 : BOOL;
    Z1 AT %IX104.4 : BOOL;
    X2 AT %IX104.5 : BOOL;
    Z2 AT %IX104.6 : BOOL;
    X3 AT %IX104.7 : BOOL;
    Z3 AT %IX105.0 : BOOL;
    Liift AT %QX110.3 : BOOL;
    Leeft AT %QX110.4 : BOOL;
    Riight AT %QX110.5 : BOOL;
    Liift2 AT %QX110.6 : BOOL;
    Leeft2 AT %QX110.7 : BOOL;
    Riight2 AT %QX111.0 : BOOL;
    Liift3 AT %QX111.1 : BOOL;
    Leeft3 AT %QX111.2 : BOOL;
    Riight3 AT %QX111.3 : BOOL;
    LoadCon1 AT %QX111.4 : BOOL;
    LoadCon2 AT %QX111.5 : BOOL;
    LoadCon3 AT %QX111.6 : BOOL;
    LoadCon4 AT %QX111.7 : BOOL;
    LoadCon5 AT %QX112.0 : BOOL;
    Target AT %QW106 : INT;
    Target2 AT %QW107 : INT;
    Target3 AT %QW108 : INT;
    DIGDIS1 AT %QW109 : INT;
    DIGDIS2 AT %QW110 : INT;
    DIGDIS3 AT %QW111 : INT;
    VIR1 AT %QX4.3 : BOOL;
    VIR2 AT %QX4.4 : BOOL;
    VIR3 AT %QX4.5 : BOOL;
    VIR4 AT %QX4.6 : BOOL;
    VIR5 AT %QX4.7 : BOOL;
    VIR6 AT %QX5.3 : BOOL;
    VIRblckx1 AT %QX5.0 : BOOL;
    VIRblckz1 AT %QX5.1 : BOOL;
    Hijau AT %QX5.2 : BOOL;
    Switch1 AT %QX5.4 : BOOL;
    Reset1 AT %QX5.5 : BOOL;
    VIR7 AT %QX6.0 : BOOL;
    VIR8 AT %QX6.1 : BOOL;
    VIR9 AT %QX6.2 : BOOL;
    VIR10 AT %QX6.3 : BOOL;
    VIR11 AT %QX6.4 : BOOL;
    VIR12 AT %QX6.5 : BOOL;
    VIRblckx2 AT %QX6.6 : BOOL;
    VIRblckz2 AT %QX6.7 : BOOL;
    Metal AT %QX7.0 : BOOL;
    Switch2 AT %QX7.1 : BOOL;
    Reset2 AT %QX7.2 : BOOL;
    VIR13 AT %QX7.3 : BOOL;
    VIR14 AT %QX7.4 : BOOL;
    VIR15 AT %QX7.5 : BOOL;
    VIR16 AT %QX7.6 : BOOL;
    VIR17 AT %QX7.7 : BOOL;
    VIRblckx3 AT %QX8.0 : BOOL;
    VIRblckz3 AT %QX8.1 : BOOL;
    Switch3 AT %QX8.2 : BOOL;
    Reset3 AT %QX8.3 : BOOL;
    VR1 AT %QX8.6 : BOOL;
  END_VAR
  VAR
    TON0 : TON;
    TON1 : TON;
    CTU0 : CTU;
    TON2 : TON;
    TON7 : TON;
    TON4 : TON;
    TON6 : TON;
    TON3 : TON;
    CTU1 : CTU;
    TON5 : TON;
    TON8 : TON;
    TON9 : TON;
    TON10 : TON;
    TON11 : TON;
    TON12 : TON;
    TON13 : TON;
    CTU2 : CTU;
    TON14 : TON;
    TON15 : TON;
    TON16 : TON;
    TON17 : TON;
    TON18 : TON;
    TON19 : TON;
    TON20 : TON;
    CTU3 : CTU;
    TON21 : TON;
    TON22 : TON;
    TON23 : TON;
    TON24 : TON;
    TON25 : TON;
    CTU4 : CTU;
    TON26 : TON;
    TON27 : TON;
    TON28 : TON;
    TON29 : TON;
    TON30 : TON;
    CTU5 : CTU;
    CTU6 : CTU;
  END_VAR
  VAR  (* added by the conversion: wires and edge detectors of the diagram *)
    R_TRIG1 : R_TRIG;
    R_TRIG2 : R_TRIG;
    F_TRIG3 : F_TRIG;
    F_TRIG4 : F_TRIG;
    F_TRIG5 : F_TRIG;
    R_TRIG6 : R_TRIG;
    F_TRIG7 : F_TRIG;
    F_TRIG8 : F_TRIG;
    R_TRIG9 : R_TRIG;
    F_TRIG10 : F_TRIG;
    _AND69_OUT : BOOL;
    _AND190_OUT : BOOL;
    F_TRIG11 : F_TRIG;
    R_TRIG12 : R_TRIG;
    R_TRIG13 : R_TRIG;
    R_TRIG14 : R_TRIG;
    F_TRIG15 : F_TRIG;
    F_TRIG16 : F_TRIG;
    R_TRIG17 : R_TRIG;
    F_TRIG18 : F_TRIG;
    _AND290_OUT : BOOL;
  END_VAR

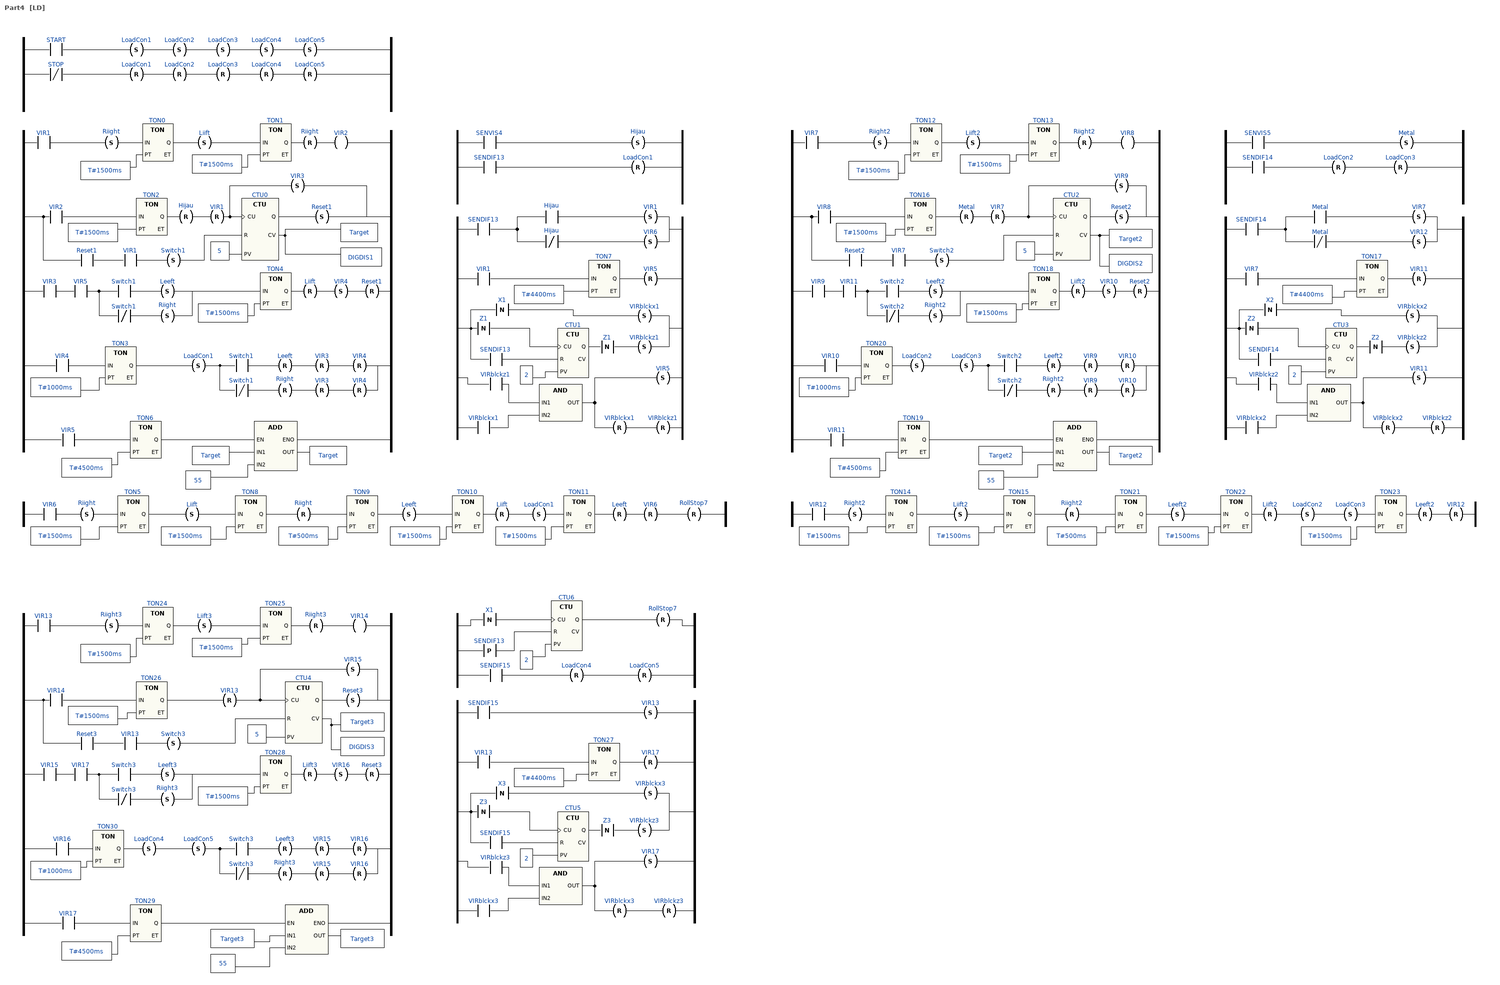
(* LD diagram, written out as Structured Text *)
IF START THEN LoadCon1 := TRUE; END_IF;
IF START THEN LoadCon2 := TRUE; END_IF;
IF START THEN LoadCon3 := TRUE; END_IF;
IF START THEN LoadCon4 := TRUE; END_IF;
IF START THEN LoadCon5 := TRUE; END_IF;
IF NOT STOP THEN LoadCon1 := FALSE; END_IF;
IF NOT STOP THEN LoadCon2 := FALSE; END_IF;
IF NOT STOP THEN LoadCon3 := FALSE; END_IF;
IF NOT STOP THEN LoadCon4 := FALSE; END_IF;
IF NOT STOP THEN LoadCon5 := FALSE; END_IF;
IF VIR1 THEN Riight := TRUE; END_IF;
TON0(IN := VIR1, PT := T#1500ms);
IF TON0.Q THEN Liift := TRUE; END_IF;
TON1(IN := TON0.Q, PT := T#1500ms);
IF TON1.Q THEN Riight := FALSE; END_IF;
VIR2 := TON1.Q;
IF SENVIS4 THEN Hijau := TRUE; END_IF;
IF VIR7 THEN Riight2 := TRUE; END_IF;
TON12(IN := VIR7, PT := T#1500ms);
IF TON12.Q THEN Liift2 := TRUE; END_IF;
TON13(IN := TON12.Q, PT := T#1500ms);
IF TON13.Q THEN Riight2 := FALSE; END_IF;
VIR8 := TON13.Q;
IF SENVIS5 THEN Metal := TRUE; END_IF;
IF SENDIF13 THEN LoadCon1 := FALSE; END_IF;
IF SENDIF14 THEN LoadCon2 := FALSE; END_IF;
IF SENDIF14 THEN LoadCon3 := FALSE; END_IF;
TON2(IN := VIR2, PT := T#1500ms);
IF TON2.Q THEN VIR3 := TRUE; END_IF;
TON16(IN := VIR8, PT := T#1500ms);
IF TON16.Q THEN VIR9 := TRUE; END_IF;
IF TON2.Q THEN Hijau := FALSE; END_IF;
IF TON2.Q THEN VIR1 := FALSE; END_IF;
R_TRIG1(CLK := TON2.Q);
CTU0(CU := R_TRIG1.Q, R := Reset1 AND VIR1, PV := 5);
IF CTU0.Q THEN Reset1 := TRUE; END_IF;
IF SENDIF13 AND Hijau THEN VIR1 := TRUE; END_IF;
IF TON16.Q THEN Metal := FALSE; END_IF;
IF TON16.Q THEN VIR7 := FALSE; END_IF;
R_TRIG2(CLK := TON16.Q);
CTU2(CU := R_TRIG2.Q, R := Reset2 AND VIR7, PV := 5);
IF CTU2.Q THEN Reset2 := TRUE; END_IF;
IF SENDIF14 AND Metal THEN VIR7 := TRUE; END_IF;
Target := CTU0.CV;
Target2 := CTU2.CV;
IF SENDIF13 AND NOT Hijau THEN VIR6 := TRUE; END_IF;
IF SENDIF14 AND NOT Metal THEN VIR12 := TRUE; END_IF;
DIGDIS1 := CTU0.CV;
IF Reset1 AND VIR1 THEN Switch1 := TRUE; END_IF;
IF Reset2 AND VIR7 THEN Switch2 := TRUE; END_IF;
DIGDIS2 := CTU2.CV;
TON7(IN := VIR1, PT := T#4400ms);
IF TON7.Q THEN VIR5 := FALSE; END_IF;
TON17(IN := VIR7, PT := T#4400ms);
IF TON17.Q THEN VIR11 := FALSE; END_IF;
IF VIR3 AND VIR5 AND Switch1 THEN Leeft := TRUE; END_IF;
TON4(IN := VIR3 AND VIR5 AND (NOT Switch1 OR Switch1), PT := T#1500ms);
IF TON4.Q THEN Liift := FALSE; END_IF;
IF TON4.Q THEN VIR4 := TRUE; END_IF;
IF TON4.Q THEN Reset1 := FALSE; END_IF;
IF VIR9 AND VIR11 AND Switch2 THEN Leeft2 := TRUE; END_IF;
TON18(IN := VIR9 AND VIR11 AND (NOT Switch2 OR Switch2), PT := T#1500ms);
IF TON18.Q THEN Liift2 := FALSE; END_IF;
IF TON18.Q THEN VIR10 := TRUE; END_IF;
IF TON18.Q THEN Reset2 := FALSE; END_IF;
IF VIR3 AND VIR5 AND NOT Switch1 THEN Riight := TRUE; END_IF;
F_TRIG3(CLK := X1);
IF F_TRIG3.Q THEN VIRblckx1 := TRUE; END_IF;
IF VIR9 AND VIR11 AND NOT Switch2 THEN Riight2 := TRUE; END_IF;
F_TRIG4(CLK := X2);
IF F_TRIG4.Q THEN VIRblckx2 := TRUE; END_IF;
F_TRIG5(CLK := Z1);
R_TRIG6(CLK := F_TRIG5.Q);
CTU1(CU := R_TRIG6.Q, R := SENDIF13, PV := 2);
F_TRIG7(CLK := Z1);
IF CTU1.Q AND F_TRIG7.Q THEN VIRblckz1 := TRUE; END_IF;
F_TRIG8(CLK := Z2);
R_TRIG9(CLK := F_TRIG8.Q);
CTU3(CU := R_TRIG9.Q, R := SENDIF14, PV := 2);
F_TRIG10(CLK := Z2);
IF CTU3.Q AND F_TRIG10.Q THEN VIRblckz2 := TRUE; END_IF;
TON3(IN := VIR4, PT := T#1000ms);
IF TON3.Q THEN LoadCon1 := TRUE; END_IF;
IF TON3.Q AND Switch1 THEN Leeft := FALSE; END_IF;
IF TON3.Q AND Switch1 THEN VIR3 := FALSE; END_IF;
IF TON3.Q AND Switch1 THEN VIR4 := FALSE; END_IF;
TON20(IN := VIR10, PT := T#1000ms);
IF TON20.Q THEN LoadCon2 := TRUE; END_IF;
IF TON20.Q THEN LoadCon3 := TRUE; END_IF;
IF TON20.Q AND Switch2 THEN Leeft2 := FALSE; END_IF;
IF TON20.Q AND Switch2 THEN VIR9 := FALSE; END_IF;
IF TON20.Q AND Switch2 THEN VIR10 := FALSE; END_IF;
_AND69_OUT := VIRblckz1 AND VIRblckx1;
IF _AND69_OUT THEN VIR5 := TRUE; END_IF;
_AND190_OUT := VIRblckz2 AND VIRblckx2;
IF _AND190_OUT THEN VIR11 := TRUE; END_IF;
IF TON3.Q AND NOT Switch1 THEN Riight := FALSE; END_IF;
IF TON3.Q AND NOT Switch1 THEN VIR3 := FALSE; END_IF;
IF TON3.Q AND NOT Switch1 THEN VIR4 := FALSE; END_IF;
IF TON20.Q AND NOT Switch2 THEN Riight2 := FALSE; END_IF;
IF TON20.Q AND NOT Switch2 THEN VIR9 := FALSE; END_IF;
IF TON20.Q AND NOT Switch2 THEN VIR10 := FALSE; END_IF;
IF _AND69_OUT THEN VIRblckx1 := FALSE; END_IF;
IF _AND69_OUT THEN VIRblckz1 := FALSE; END_IF;
IF _AND190_OUT THEN VIRblckx2 := FALSE; END_IF;
IF _AND190_OUT THEN VIRblckz2 := FALSE; END_IF;
TON6(IN := VIR5, PT := T#4500ms);
IF TON6.Q THEN Target := Target + 55; END_IF;
TON19(IN := VIR11, PT := T#4500ms);
IF TON19.Q THEN Target2 := Target2 + 55; END_IF;
IF VIR6 THEN Riight := TRUE; END_IF;
TON5(IN := VIR6, PT := T#1500ms);
IF TON5.Q THEN Liift := TRUE; END_IF;
TON8(IN := TON5.Q, PT := T#1500ms);
IF TON8.Q THEN Riight := FALSE; END_IF;
TON9(IN := TON8.Q, PT := T#500ms);
IF TON9.Q THEN Leeft := TRUE; END_IF;
TON10(IN := TON9.Q, PT := T#1500ms);
IF TON10.Q THEN Liift := FALSE; END_IF;
IF TON10.Q THEN LoadCon1 := TRUE; END_IF;
TON11(IN := TON10.Q, PT := T#1500ms);
IF TON11.Q THEN Leeft := FALSE; END_IF;
IF TON11.Q THEN VIR6 := FALSE; END_IF;
IF TON11.Q THEN RollStop7 := FALSE; END_IF;
IF VIR12 THEN Riight2 := TRUE; END_IF;
TON14(IN := VIR12, PT := T#1500ms);
IF TON14.Q THEN Liift2 := TRUE; END_IF;
TON15(IN := TON14.Q, PT := T#1500ms);
IF TON15.Q THEN Riight2 := FALSE; END_IF;
TON21(IN := TON15.Q, PT := T#500ms);
IF TON21.Q THEN Leeft2 := TRUE; END_IF;
TON22(IN := TON21.Q, PT := T#1500ms);
IF TON22.Q THEN Liift2 := FALSE; END_IF;
IF TON22.Q THEN LoadCon2 := TRUE; END_IF;
IF TON22.Q THEN LoadCon3 := TRUE; END_IF;
TON23(IN := TON22.Q, PT := T#1500ms);
IF TON23.Q THEN Leeft2 := FALSE; END_IF;
IF TON23.Q THEN VIR12 := FALSE; END_IF;
F_TRIG11(CLK := X1);
R_TRIG12(CLK := F_TRIG11.Q);
R_TRIG13(CLK := SENDIF13);
CTU6(CU := R_TRIG12.Q, R := R_TRIG13.Q, PV := 2);
IF CTU6.Q THEN RollStop7 := FALSE; END_IF;
IF VIR13 THEN Riight3 := TRUE; END_IF;
TON24(IN := VIR13, PT := T#1500ms);
IF TON24.Q THEN Liift3 := TRUE; END_IF;
TON25(IN := TON24.Q, PT := T#1500ms);
IF TON25.Q THEN Riight3 := FALSE; END_IF;
VIR14 := TON25.Q;
TON26(IN := VIR14, PT := T#1500ms);
IF TON26.Q THEN VIR15 := TRUE; END_IF;
IF SENDIF15 THEN LoadCon4 := FALSE; END_IF;
IF SENDIF15 THEN LoadCon5 := FALSE; END_IF;
IF TON26.Q THEN VIR13 := FALSE; END_IF;
R_TRIG14(CLK := TON26.Q);
CTU4(CU := R_TRIG14.Q, R := Reset3 AND VIR13, PV := 5);
IF CTU4.Q THEN Reset3 := TRUE; END_IF;
IF SENDIF15 THEN VIR13 := TRUE; END_IF;
Target3 := CTU4.CV;
IF Reset3 AND VIR13 THEN Switch3 := TRUE; END_IF;
DIGDIS3 := CTU4.CV;
TON27(IN := VIR13, PT := T#4400ms);
IF TON27.Q THEN VIR17 := FALSE; END_IF;
IF VIR15 AND VIR17 AND Switch3 THEN Leeft3 := TRUE; END_IF;
TON28(IN := VIR15 AND VIR17 AND (NOT Switch3 OR Switch3), PT := T#1500ms);
IF TON28.Q THEN Liift3 := FALSE; END_IF;
IF TON28.Q THEN VIR16 := TRUE; END_IF;
IF TON28.Q THEN Reset3 := FALSE; END_IF;
F_TRIG15(CLK := X3);
IF F_TRIG15.Q THEN VIRblckx3 := TRUE; END_IF;
IF VIR15 AND VIR17 AND NOT Switch3 THEN Riight3 := TRUE; END_IF;
F_TRIG16(CLK := Z3);
R_TRIG17(CLK := F_TRIG16.Q);
CTU5(CU := R_TRIG17.Q, R := SENDIF15, PV := 2);
F_TRIG18(CLK := Z3);
IF CTU5.Q AND F_TRIG18.Q THEN VIRblckz3 := TRUE; END_IF;
TON30(IN := VIR16, PT := T#1000ms);
IF TON30.Q THEN LoadCon4 := TRUE; END_IF;
IF TON30.Q THEN LoadCon5 := TRUE; END_IF;
IF TON30.Q AND Switch3 THEN Leeft3 := FALSE; END_IF;
IF TON30.Q AND Switch3 THEN VIR15 := FALSE; END_IF;
IF TON30.Q AND Switch3 THEN VIR16 := FALSE; END_IF;
_AND290_OUT := VIRblckz3 AND VIRblckx3;
IF _AND290_OUT THEN VIR17 := TRUE; END_IF;
IF TON30.Q AND NOT Switch3 THEN Riight3 := FALSE; END_IF;
IF TON30.Q AND NOT Switch3 THEN VIR15 := FALSE; END_IF;
IF TON30.Q AND NOT Switch3 THEN VIR16 := FALSE; END_IF;
IF _AND290_OUT THEN VIRblckx3 := FALSE; END_IF;
IF _AND290_OUT THEN VIRblckz3 := FALSE; END_IF;
TON29(IN := VIR17, PT := T#4500ms);
IF TON29.Q THEN Target3 := Target3 + 55; END_IF;
END_PROGRAM

CONFIGURATION Config0
  RESOURCE Res0 ON PLC
    VAR_GLOBAL
      START AT %IX100.0 : BOOL;
      STOP AT %IX100.1 : BOOL;
      SENDIF13 AT %IX103.6 : BOOL;
      CONR4_1 AT %QX108.1 : BOOL;
      CONR4_2 AT %QX108.2 : BOOL;
      CON6_3 AT %QX101.2 : BOOL;
      CON6_5 AT %QX101.4 : BOOL;
      CON6_7 AT %QX101.6 : BOOL;
      RollStop7 AT %QX112.1 : BOOL;
    END_VAR
    TASK task0(INTERVAL := T#20ms, PRIORITY := 0);
    TASK task1(INTERVAL := T#20ms, PRIORITY := 0);
    TASK task2(INTERVAL := T#20ms, PRIORITY := 0);
    TASK task3(INTERVAL := T#20ms, PRIORITY := 0);
    PROGRAM instance0 WITH task0 : Part1;
    PROGRAM instance1 WITH task1 : Part2;
    PROGRAM instance2 WITH task2 : Part3;
    PROGRAM instance3 WITH task3 : Part4;
  END_RESOURCE
END_CONFIGURATION
